// Mitsubishi GX Works2 project: 电动机循环启动   PLC: FX3U/FX3UC

PROGRAM MAIN
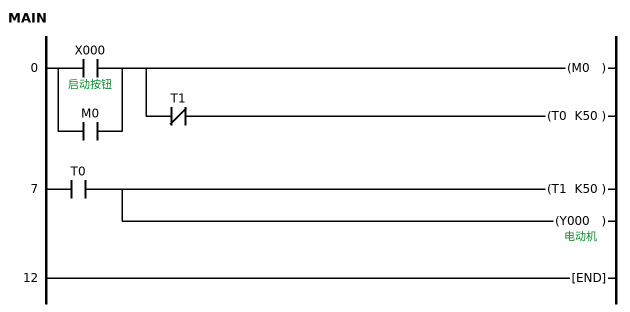
0     LD      X000  ; 启动按钮
      OR      M0
      OUT     M0
      ANI     T1
      OUT     T0 K50
7     LD      T0
      OUT     T1 K50
      OUT     Y000  ; 电动机
12    END
END_PROGRAM

// device comments not shown above
X001  ; 关闭按钮
